(* Manages and scales all analog inputs *)

PROGRAM Analog_Manager
  VAR_EXTERNAL
    Level : REAL;
    Temperature : REAL;
    Pressure : REAL;
    Weight : REAL;
  END_VAR
  VAR
    Raw_Level : REAL;
    Raw_Temperature : REAL;
    Raw_Pressure : REAL;
    Raw_Weight : REAL;
  END_VAR

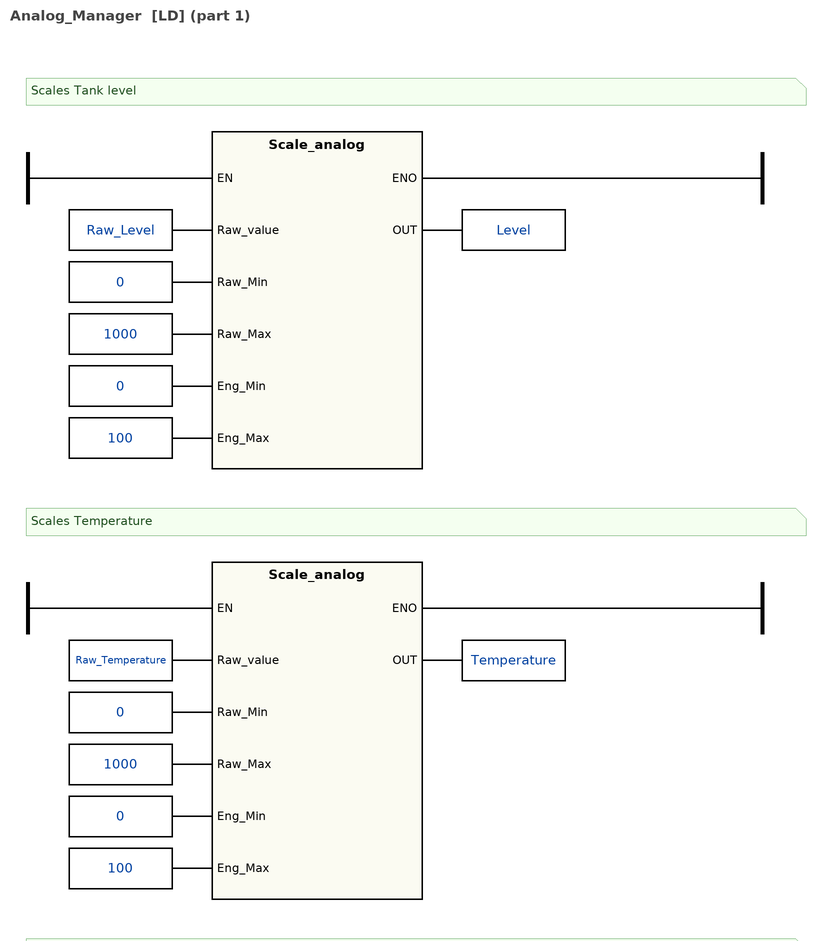
(* LD diagram, written out as Structured Text *)
(* Scales Tank level *)
Level := Scale_analog(Raw_Level, 0, 1000, 0, 100);
(* Scales Temperature *)
Temperature := Scale_analog(Raw_Temperature, 0, 1000, 0, 100);
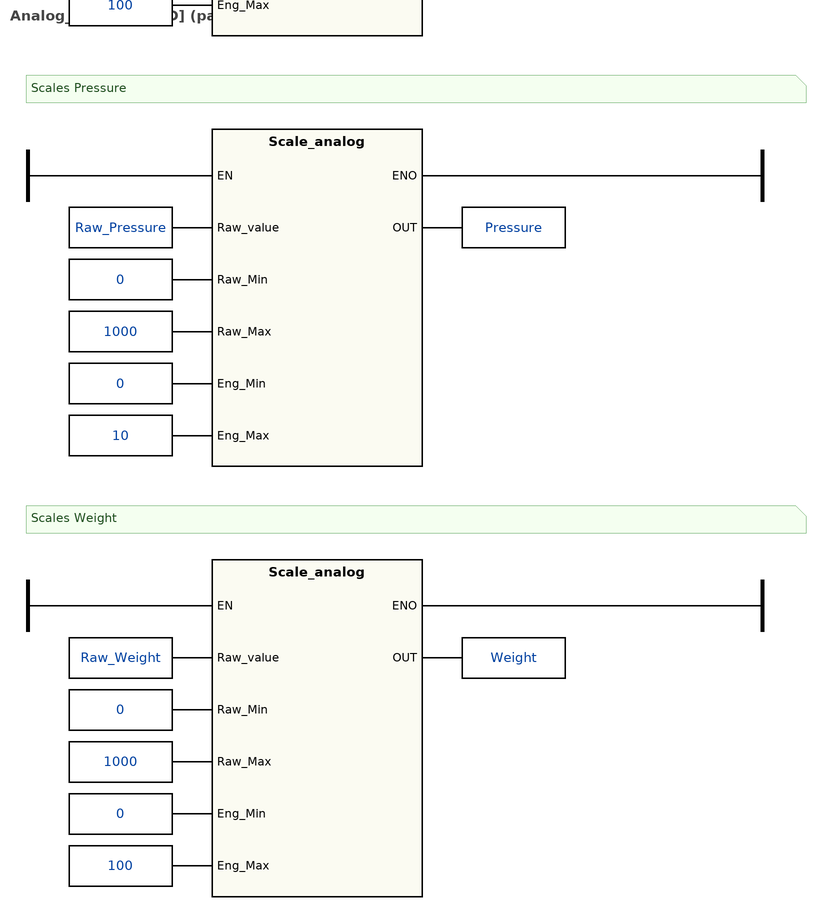
(* Scales Pressure *)
Pressure := Scale_analog(Raw_Pressure, 0, 1000, 0, 10);
(* Scales Weight *)
Weight := Scale_analog(Raw_Weight, 0, 1000, 0, 100);
END_PROGRAM
